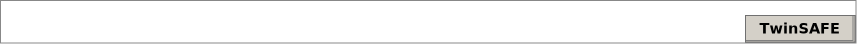
VISUALIZATION AX5805_Specific_Diagnostics  // 857x44
    Button (745,15 110x27), "TwinSAFE"
        OnMouseClick: change screen: TwinSAFE
        OnMouseUp: execute { g_xHMI_ErrAckPB := FALSE ; }
END_VISUALIZATION

(* stored: Version 1.1.0.1, ProductVersion 3.1.0.18
   Visu AX5805_Specific_Diagnostics: Id {681d1355-4aa0-4d1b-957b-a9e99484e672} *)
